ADAPTER IAS_Skill
  (* Standard: 61499-1 *)
  (* Version 0.0, 2008-04-22, GE, 4DIAC-Consortium *)
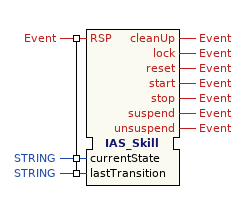
  EVENT_INPUT
    RSP WITH currentState, lastTransition;
  END_EVENT
  EVENT_OUTPUT
    cleanUp;
    lock;
    reset;
    start;
    stop;
    suspend;
    unsuspend;
  END_EVENT
  VAR_INPUT
    currentState : STRING;
    lastTransition : STRING;
  END_VAR
  SERVICE SOCKET/PLUG
    SEQUENCE normal_operation
      PLUG.start() -> SOCKET.start();
      SOCKET.RSP(currentState="Executing") -> PLUG.RSP(currentState="Executing");
      SOCKET.RSP(currentState="Idle") -> PLUG.RSP(currentState="Idle");
    END_SEQUENCE
    SEQUENCE indication_response
    END_SEQUENCE
    SEQUENCE error_handling (* should be executed if an error occurs *)
      PLUG.reset() -> SOCKET.reset();
      SOCKET.RSP(currentState="Idle") -> PLUG.RSP(currentState="Idle");
    END_SEQUENCE
    SEQUENCE error_signal
      SOCKET.RSP(currentState="Locked") -> PLUG.RSP(currentState="Locked");
    END_SEQUENCE
  END_SERVICE
END_ADAPTER
